(* IEC 61131-3 sources: moqui-plc/agent-skills/output/sessions/tank-level-control-001/generated-plc/codesys-applications/TankLevelControl/runtime/component/main/src/main/mantle/main, 3 files *)

(* ---- MainStatus.dut ---- *)
{attribute 'qualified_only'}
{attribute 'strict'}
TYPE MainStatus : (
    Standby := 0,
    Run,
    Fault
); END_TYPE

(* Questions for the skill/user:
 * 1. Which StatusFlow is used for the main orchestration FSM?
 * 2. In which order should the states appear in the enum?
 * 3. Which state is the initial steady state?
 * 4. Which state is the fault state?
 *
 * Generation note:
 * - This enum is typically derived from StatusFlowItem entries related to the selected main StatusFlow.
 * - The generated names should match the identifiers used by Main.pou and MainRuleEngine.pou.
 *)

(* ---- Main.pou ---- *)
{attribute 'no_assign'}
(*
 * NOTE: In general, the Main component implements the control logic of automated industrial systems (Finite State Machine - FSM)
 * using hierarchical control architectures. It separates control policies from implementation mechanisms,
 * and diagnostic mechanisms from failure/error reaction and system reset policies.
 *
 * MainRuleEngine generates transition requests; Main consumes them.
 * DeviceManager orchestrates the individual device FBs.
 *
 * Call order in the PLC task:
 *   InputSignalUpdate -> Main -> DeviceManager -> OutputSignalUpdate
 *)
FUNCTION_BLOCK Main
VAR_EXTERNAL
    dev : DeviceFacade;
    workEffort : WorkEffort;
END_VAR
VAR_INPUT
    operationType : OperatingMode;
    enable : BOOL;
END_VAR
VAR_OUTPUT
    done : BOOL;
    error : BOOL;
END_VAR
VAR CONSTANT
    componentName : STRING := 'main';
END_VAR
VAR
    (* Logger facade *)
    logger : LoggerFacade;
    (* FSM transition logic *)
    ruleEngine : MainRuleEngine;
    (* No subsystem controllers. *)
    (* HAL manager *)
    deviceManager : DeviceManager;
END_VAR

(* Logger facade init *)
logger.enable := TRUE; logger.loggerName := componentName;

IF NOT enable THEN RETURN; END_IF;

(* Init: device setup and configuration *)
IF (operationType = OperatingMode.Init) THEN
    logger(message := 'Setup and configuration of all devices.', level := LogLevel.DEBUG);
    (* The static device configuration parameters are mapped directly by the device config manager (recipe manager),
     * while only the dynamic parameters are mapped below in the standby status.
     *)
    (* Reset signal manager *)
    dev.signalMgmt(operationType := SignalMgmtOperatingMode.Reset, loggerName := componentName);
    dev.status := MainStatus.Standby;
    dev.lastStatus := MainStatus.Standby;
    done := FALSE;
    ; (* no additional project-specific initialization *)
    (* No subsystem controller initialization. *)
ELSE
    (* FSM transition-condition rule engine *)
    logger(message := 'Run FSM transition-condition logic.', level := LogLevel.DEBUG);
    ruleEngine(operationType := operationType);
END_IF;

dev.lastStatus := dev.status;

(* Optional fault-state override; emitted only when the reviewed FSM defines one. *)
IF dev.faultRequest THEN dev.status := MainStatus.Fault; END_IF;

(* Main FSM - Output function + State-update function *)
logger(message := 'Run Main FSM.', level := LogLevel.DEBUG);
CASE dev.status OF
    MainStatus.Standby :
        logger(message := 'Standby.', level := LogLevel.DEBUG);

        (* FSM output function *)
        dev.levelControllerEnable := FALSE;
        dev.levelControllerOutputFreezeEnable := FALSE; (* No freeze needed while the PID is disabled. *)
        dev.levelControllerValveOut := 0.0; (* Safe default: valve closed while stopped (confirmed). *)

        (* FSM status update function *)
        IF dev.runRequest THEN
            (* Start -> Run *)
            dev.status := MainStatus.Run;
        END_IF;

    MainStatus.Run :
        logger(message := 'Run.', level := LogLevel.DEBUG);

        (* FSM output function *)
        dev.levelControllerEnable := TRUE;
        dev.levelControllerOutputFreezeEnable := FALSE; (* Normal automatic modulation. *)
        dev.levelControllerValveOut := dev.levelControllerOutputActual; (* PID drives the valve directly. *)

        (* FSM status update function *)
        IF dev.standbyRequest THEN
            (* Stop -> Standby *)
            dev.status := MainStatus.Standby;
        END_IF;

    MainStatus.Fault :
        logger(message := 'Fault.', level := LogLevel.DEBUG);

        (* FSM output function *)
        dev.levelControllerEnable := TRUE;
        dev.levelControllerOutputFreezeEnable := TRUE; (* Generic-fault recommendation: keep PID alive but freeze output at the last computed value using the native ProcessPid outputFreezeEnable input (no external latch needed). *)
        dev.levelControllerValveOut := SEL(dev.levelLL, SEL(dev.levelHH, dev.levelControllerOutputActual, 0.0), 100.0); (* LL forces the valve open (100%, avoid running the tank dry); HH forces the valve closed (0%, avoid overflow); otherwise (e.g. LT sensor out-of-range) hold the frozen PID output. SEL(G,IN0, IN1) returns IN1 when G is TRUE, IN0 otherwise. *)

        (* FSM status update function *)
        IF dev.standbyRequest THEN
            (* AutoRecover -> Standby *)
            dev.status := MainStatus.Standby;
        END_IF;
END_CASE;

(* Subsystem FSMs execute after the supervisor output/state update and before the HAL. *)
(* No subsystem controller calls. *)

done := FALSE;

(* Device orchestration (HAL) *)
logger(message := 'Update devices.', level := LogLevel.DEBUG);
deviceManager(operationType := operationType);

(* ---- MainRuleEngine.pou ---- *)
{attribute 'no_assign'}
(*
 * MainRuleEngine - transition-condition logic for the supervisor FSM.
 *
 * Responsibilities:
 *   1. Reset transition requests to safe defaults.
 *   2. Run the signal management engine (fault / alarm / warning detection).
 *   3. Compute boolean predicates from sensor feedback and recipe setpoints.
 *   4. Implement the per-state transition-condition rules.
 *
 * Requests are reset every scan. A state persists until a reviewed transition
 * condition asserts the corresponding request consumed by Main.
 *)
FUNCTION_BLOCK MainRuleEngine
VAR_EXTERNAL
    clks : Clocks;
    dev : DeviceFacade;
    workEffort : WorkEffort;
END_VAR
VAR_INPUT
    operationType : OperatingMode := OperatingMode.Run;
END_VAR
VAR_OUTPUT
    error : BOOL;
END_VAR
VAR
    (* Device diagnostics *)
    deviceDiags : DeviceDiagnostics;
END_VAR

(* Reset transition requests to FALSE before evaluating transition policy. *)
dev.faultRequest := FALSE;
dev.standbyRequest := FALSE;
dev.runRequest := FALSE;

deviceDiags(operationType := operationType, error => error);

(* Compute sensor predicates *)
dev.levelLL := dev.levelControllerLevelIn <= dev.levelControllerLevelLowLowThreshold; (* Low-Low level alarm (threshold confirmed by developer: 5%). *)
dev.levelHH := dev.levelControllerLevelIn >= dev.levelControllerLevelHighHighThreshold; (* High-High level alarm (threshold confirmed by developer: 95%). *)
dev.levelSensorFault := (dev.levelControllerLevelIn < -2.0) OR (dev.levelControllerLevelIn > 102.0); (* LT broken-wire/out-of-range detection, standard convention for a 4-20mA input scaled to 0-100%. Generic-fault trigger, per developer choice. *)

(* Fault gate *)
IF dev.levelLL OR dev.levelHH OR dev.levelSensorFault THEN
    dev.faultRequest := TRUE;
    RETURN;
END_IF;

(* Transition-condition rule engine. Conditions are evaluated by precedence. *)
CASE dev.status OF
    MainStatus.Standby :
        (* State Standby transition conditions *)
        IF dev.levelControllerRunCmd THEN
            (* Start -> Run *)
            dev.runRequest := TRUE;
        END_IF;

    MainStatus.Run :
        (* State Run transition conditions *)
        IF NOT dev.levelControllerRunCmd THEN
            (* Stop -> Standby *)
            dev.standbyRequest := TRUE;
        END_IF;

    MainStatus.Fault :
        (* State Fault transition conditions *)
        IF TRUE THEN
            (* AutoRecover -> Standby *)
            dev.standbyRequest := TRUE;
        END_IF;
END_CASE;
